{attribute 'OPC.UA.DA.StructuredType' := '1'}
TYPE SBoolExpressionSpec :
STRUCT
	Operator: EBoolOperation;
	
	LeftType: EExpressionType;
	LeftIdx: UINT;
	
	RightType: EExpressionType;
	RightIdx: UINT;
END_STRUCT
END_TYPE

(* stored: Version 1.1.0.1
   DUT SBoolExpressionSpec: Id {465cf94a-d301-40e7-b5e3-a603d00f70bb} *)
